// TIA Portal V20 export
VAR_GLOBAL   // PLC tag table "Unit1Em10"
   "BA060ZSIBK17.00" AT %I1064.0 : Bool;   // (HOME) LASER MARKING COVER UP
   "BA060ZSIBK17.01" AT %I1064.1 : Bool;   // (WORK) LASER MARKING COVER DOWN
   "BA060ZSIBK17.02" AT %I1064.2 : Bool;   // (WORK) LASER MARKING Stage Lift UP
   "BA060ZSIBK17.03" AT %I1064.3 : Bool;   // (HOME) LASER MARKING Stage Lift DOWN
   "BA060ZSIBK17.06" AT %I1064.6 : Bool;   // SPARE
   "BA060ZSIBK17.05" AT %I1064.5 : Bool;   // LASER MARKING STACK DETECT SENSOR
   "BA060ZSIBK17.04" AT %I1064.4 : Bool;   // SPARE
   "BA060ZSIBK17.07" AT %I1064.7 : Bool;   // SPARE
   "BA060ZSIPM09.04" AT %Q2032.4 : Bool;   // (HOME) LASER MARKING COVER UP
   "BA060ZSIPM09.05" AT %Q2032.5 : Bool;   // (WORK) LASER MARKING COVER DOWN
   "BA060ZSIPM09.06" AT %Q2032.6 : Bool;   // (WORK) LASER MARKING STAGE LIFT UP
   "BA060ZSIPM09.07" AT %Q2032.7 : Bool;   // (HOME) LASER MARKING STAGE LIFT DOWN
   "BA060AZSISP504.04" AT %Q3000.4 : Bool;   // QR MARKING TRIGGER IN
   "BA060AZSISP504.05" AT %Q3000.5 : Bool;   // SPARE
   "BA060AZSISP504.06" AT %Q3000.6 : Bool;   // SPARE
   "BA060AZSISP504.07" AT %Q3000.7 : Bool;   // SPARE
END_VAR
VAR_GLOBAL CONSTANT   // user constants
   U1EM10_JOB01 : DInt := 1;
   U1EM10_JOB02 : DInt := 2;
   U1EM10_JOB03 : DInt := 3;
   U1EM10_JOB04 : DInt := 4;
   U1EM10_JOB05 : DInt := 5;
   U1EM10_JOB06 : DInt := 6;
   U1EM10_JOB07 : DInt := 7;
   U1EM10_JOB08 : DInt := 8;
   U1EM10_JOB09 : DInt := 9;
   U1EM10_JOB10 : DInt := 10;
   U1EM10_JOB11 : DInt := 11;
   U1EM10_JOB12 : DInt := 12;
   U1EM10_JOB13 : DInt := 13;
   U1EM10_JOB14 : DInt := 14;
   U1EM10_JOB15 : DInt := 15;
   U1EM10_JOB16 : DInt := 16;
   U1EM10_JOB17 : DInt := 17;
   U1EM10_JOB18 : DInt := 18;
   U1EM10_JOB19 : DInt := 19;
   U1EM10_JOB20 : DInt := 20;
   U1EM10_JOB21 : DInt := 21;
   U1EM10_JOB22 : DInt := 22;
   U1EM10_JOB23 : DInt := 23;
   U1EM10_JOB24 : DInt := 24;
   U1EM10_JOB25 : DInt := 25;
   U1EM10_JOB26 : DInt := 26;
   U1EM10_JOB27 : DInt := 27;
   U1EM10_JOB28 : DInt := 28;
   U1EM10_JOB29 : DInt := 29;
   U1EM10_JOB30 : DInt := 30;
   U1EM10_JOB31 : DInt := 31;
   U1EM10_JOB32 : DInt := 32;
   U1EM10_JOB33 : DInt := 33;
   U1EM10_JOB34 : DInt := 34;
   U1EM10_JOB35 : DInt := 35;
   U1EM10_JOB36 : DInt := 36;
   U1EM10_JOB37 : DInt := 37;
   U1EM10_JOB38 : DInt := 38;
   U1EM10_JOB39 : DInt := 39;
   U1EM10_JOB40 : DInt := 40;
   U1EM10_JOB41 : DInt := 41;
   U1EM10_JOB42 : DInt := 42;
   U1EM10_JOB43 : DInt := 43;
   U1EM10_JOB44 : DInt := 44;
   U1EM10_JOB45 : DInt := 45;
   U1EM10_JOB46 : DInt := 46;
   U1EM10_JOB47 : DInt := 47;
   U1EM10_JOB48 : DInt := 48;
   U1EM10_JOB49 : DInt := 49;
   U1EM10_JOB50 : DInt := 50;
   U1EM10_JOB51 : DInt := 51;
   U1EM10_JOB52 : DInt := 52;
   U1EM10_JOB53 : DInt := 53;
   U1EM10_JOB54 : DInt := 54;
   U1EM10_JOB55 : DInt := 55;
   U1EM10_JOB56 : DInt := 56;
   U1EM10_JOB57 : DInt := 57;
   U1EM10_JOB58 : DInt := 58;
   U1EM10_JOB59 : DInt := 59;
   U1EM10_JOB60 : DInt := 60;
   U1EM10_JOB61 : DInt := 61;
   U1EM10_JOB62 : DInt := 62;
   U1EM10_JOB63 : DInt := 63;
   U1EM10_JOB64 : DInt := 64;
   U1EM10_JOB65 : DInt := 65;
   U1EM10_JOB66 : DInt := 66;
   U1EM10_JOB67 : DInt := 67;
   U1EM10_JOB68 : DInt := 68;
   U1EM10_JOB69 : DInt := 69;
   U1EM10_JOB70 : DInt := 70;
   U1EM10_JOB71 : DInt := 71;
   U1EM10_JOB72 : DInt := 72;
   U1EM10_JOB73 : DInt := 73;
   U1EM10_JOB74 : DInt := 74;
   U1EM10_JOB75 : DInt := 75;
   U1EM10_JOB76 : DInt := 76;
   U1EM10_JOB77 : DInt := 77;
   U1EM10_JOB78 : DInt := 78;
   U1EM10_JOB79 : DInt := 79;
   U1EM10_JOB80 : DInt := 80;
   U1EM10_JOB81 : DInt := 81;
   U1EM10_JOB82 : DInt := 82;
   U1EM10_JOB83 : DInt := 83;
   U1EM10_JOB84 : DInt := 84;
   U1EM10_JOB85 : DInt := 85;
   U1EM10_JOB86 : DInt := 86;
   U1EM10_JOB87 : DInt := 87;
   U1EM10_JOB88 : DInt := 88;
   U1EM10_JOB89 : DInt := 89;
   U1EM10_JOB90 : DInt := 90;
   U1EM10_JOB91 : DInt := 91;
   U1EM10_JOB92 : DInt := 92;
   U1EM10_JOB93 : DInt := 93;
   U1EM10_JOB94 : DInt := 94;
   U1EM10_JOB95 : DInt := 95;
   U1EM10_JOB96 : DInt := 96;
   U1EM10_JOB97 : DInt := 97;
   U1EM10_JOB98 : DInt := 98;
   U1EM10_JOB99 : DInt := 99;
   U1EM10_SEQUENCE01 : Int := 1;
   U1EM10_SEQUENCE02 : Int := 2;
   U1EM10_SEQUENCE03 : Int := 3;
   U1EM10_SEQUENCE04 : Int := 4;
   U1EM10_SEQUENCE05 : Int := 5;
   U1EM10_SEQUENCE06 : Int := 6;
   U1EM10_SEQUENCE07 : Int := 7;
   U1EM10_SEQUENCE08 : Int := 8;
   U1EM10_SEQUENCE09 : Int := 9;
   U1EM10_SEQUENCE10 : Int := 10;
   U1EM10_SEQUENCE11 : Int := 11;
   U1EM10_SEQUENCE12 : Int := 12;
   U1EM10_SEQUENCE13 : Int := 13;
   U1EM10_SEQUENCE14 : Int := 14;
   U1EM10_SEQUENCE15 : Int := 15;
   U1EM10_SEQUENCE16 : Int := 16;
   U1EM10_SEQUENCE17 : Int := 17;
   U1EM10_SEQUENCE18 : Int := 18;
   U1EM10_SEQUENCE19 : Int := 19;
   U1EM10_SEQUENCE20 : Int := 20;
   U1EM10_SEQUENCE21 : Int := 21;
   U1EM10_SEQUENCE22 : Int := 22;
   U1EM10_SEQUENCE23 : Int := 23;
   U1EM10_SEQUENCE24 : Int := 24;
   U1EM10_SEQUENCE25 : Int := 25;
   U1EM10_SEQUENCE26 : Int := 26;
   U1EM10_SEQUENCE27 : Int := 27;
   U1EM10_SEQUENCE28 : Int := 28;
   U1EM10_SEQUENCE29 : Int := 29;
   U1EM10_SEQUENCE30 : Int := 30;
   U1EM10_SEQUENCE31 : Int := 31;
   U1EM10_SEQUENCE32 : Int := 32;
   U1EM10_SEQUENCE33 : Int := 33;
   U1EM10_SEQUENCE34 : Int := 34;
   U1EM10_SEQUENCE35 : Int := 35;
   U1EM10_SEQUENCE36 : Int := 36;
   U1EM10_SEQUENCE37 : Int := 37;
   U1EM10_SEQUENCE38 : Int := 38;
   U1EM10_SEQUENCE39 : Int := 39;
   U1EM10_SEQUENCE40 : Int := 40;
   U1EM10_SEQUENCE41 : Int := 41;
   U1EM10_SEQUENCE42 : Int := 42;
   U1EM10_SEQUENCE43 : Int := 43;
   U1EM10_SEQUENCE44 : Int := 44;
   U1EM10_SEQUENCE45 : Int := 45;
   U1EM10_SEQUENCE46 : Int := 46;
   U1EM10_SEQUENCE47 : Int := 47;
   U1EM10_SEQUENCE48 : Int := 48;
   U1EM10_SEQUENCE49 : Int := 49;
   U1EM10_SEQUENCE50 : Int := 50;
   U1EM10_SEQUENCE51 : Int := 51;
   U1EM10_SEQUENCE52 : Int := 52;
   U1EM10_SEQUENCE53 : Int := 53;
   U1EM10_SEQUENCE54 : Int := 54;
   U1EM10_SEQUENCE55 : Int := 55;
   U1EM10_SEQUENCE56 : Int := 56;
   U1EM10_SEQUENCE57 : Int := 57;
   U1EM10_SEQUENCE58 : Int := 58;
   U1EM10_SEQUENCE59 : Int := 59;
   U1EM10_SEQUENCE60 : Int := 60;
   U1EM10_SEQUENCE61 : Int := 61;
   U1EM10_SEQUENCE62 : Int := 62;
   U1EM10_SEQUENCE63 : Int := 63;
   U1EM10_SEQUENCE64 : Int := 64;
   U1EM10_SEQUENCE65 : Int := 65;
   U1EM10_SEQUENCE66 : Int := 66;
   U1EM10_SEQUENCE67 : Int := 67;
   U1EM10_SEQUENCE68 : Int := 68;
   U1EM10_SEQUENCE69 : Int := 69;
   U1EM10_SEQUENCE70 : Int := 70;
   U1EM10_SEQUENCE71 : Int := 71;
   U1EM10_SEQUENCE72 : Int := 72;
   U1EM10_SEQUENCE73 : Int := 73;
   U1EM10_SEQUENCE74 : Int := 74;
   U1EM10_SEQUENCE75 : Int := 75;
   U1EM10_SEQUENCE76 : Int := 76;
   U1EM10_SEQUENCE77 : Int := 77;
   U1EM10_SEQUENCE78 : Int := 78;
   U1EM10_SEQUENCE79 : Int := 79;
   U1EM10_SEQUENCE80 : Int := 80;
   U1EM10_SEQUENCE81 : Int := 81;
   U1EM10_SEQUENCE82 : Int := 82;
   U1EM10_SEQUENCE83 : Int := 83;
   U1EM10_SEQUENCE84 : Int := 84;
   U1EM10_SEQUENCE85 : Int := 85;
   U1EM10_SEQUENCE86 : Int := 86;
   U1EM10_SEQUENCE87 : Int := 87;
   U1EM10_SEQUENCE88 : Int := 88;
   U1EM10_SEQUENCE89 : Int := 89;
   U1EM10_SEQUENCE90 : Int := 90;
   U1EM10_SEQUENCE91 : Int := 91;
   U1EM10_SEQUENCE92 : Int := 92;
   U1EM10_SEQUENCE93 : Int := 93;
   U1EM10_SEQUENCE94 : Int := 94;
   U1EM10_SEQUENCE95 : Int := 95;
   U1EM10_SEQUENCE96 : Int := 96;
   U1EM10_SEQUENCE97 : Int := 97;
   U1EM10_SEQUENCE98 : Int := 98;
   U1EM10_SEQUENCE99 : Int := 99;
   U1EM10_NO_OF_AXES : USInt := 0;
   U1EM10_NO_OF_SEQUENCE : Int := 0;
END_VAR
